FUNCTION_BLOCK END_RUN
VAR_INPUT
END_VAR
VAR_OUTPUT
END_VAR
VAR
END_VAR

END_FUNCTION_BLOCK

(* stored: Version 1.1.0.1, ProductVersion 3.1.4022.18
   POU END_RUN: Id {00edb92b-fe37-4664-9a57-d0af9dbc5a2e}, SpecialFunc None *)
